// TIA Portal V19 export
DATA_BLOCK "SimulationData"   // DB44
// stored: MemoryReserve 100, Namespace Unit2
BEGIN
END_DATA_BLOCK
